Staubli VAL3: iIdent1.pgx

public program iIdent1(num& nNum[] (dimensions=1))
begin
  nNum=dioGet(iIdent1)
end
